PROGRAM Initialize
VAR
END_VAR

// we want to go to the predetermined initial position (0,0,0,0)
IF IO.EndRotationSensor THEN
	IO.MotorRotation := 0;
	IO.MotorRotationDirection := 0;
	ELSE 
		IO.MotorRotationDirection := 1;
		IO.MotorRotation := 1;
	END_IF
	IF IO.EndLiftingSensor THEN
		IO.MotorLifting := 0;
		IO.MotorLiftingDirection := 0;
	ELSE 
		IO.MotorLiftingDirection := 1;
		IO.MotorLifting := 1;
	END_IF
	IF IO.EndExtensionSensor THEN
		IO.MotorExtension := 0;
		IO.MotorExtensionDirection := 0;
	ELSE 
		IO.MotorExtensionDirection := 1;
		IO.MotorExtension := 1;
	END_IF
	IF IO.EndGripSensor THEN
		IO.MotorGrip := 0;
		IO.MotorGripDirection := 0;
	ELSE 
		IO.MotorGripDirection := 1;
		IO.MotorGrip := 1;
	END_IF
	
IF IO.EndRotationSensor AND IO.EndLiftingSensor AND IO.EndExtensionSensor AND IO.EndGripSensor THEN
	IO.Initialized := TRUE;
	//InitMotors();
END_IF

END_PROGRAM

(* stored: Version 1.1.0.1, ProductVersion 3.1.4024.13
   POU Initialize: Id {acc585e9-1428-4ae4-802a-0f449af0d289}, SpecialFunc None *)
